FUNCTION_BLOCK REAL2REAL (* Basic Function Block Type *)
  (* Standard: 61499-2 *)
  (* Version 1.0, 2006-11-14, TS, PROFACTOR GmbH *)
  (* Compiler header: package fb.rt.convert; *)
  (* Compiler Java Sun JDK >1.3 *)
  (* Compiler Cpp GNU GCC >3.0 *)
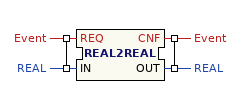
  EVENT_INPUT
    REQ WITH IN; (* Normal Execution Request *)
  END_EVENT
  EVENT_OUTPUT
    CNF WITH OUT; (* Execution Confirmation *)
  END_EVENT
  VAR_INPUT
    IN : REAL; (* Input event qualifier *)
  END_VAR
  VAR_OUTPUT
    OUT : REAL; (* Output event qualifier *)
  END_VAR
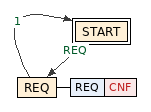
  EC_STATES
    START; (* Initial State *)
    REQ : REQ -> CNF; (* Normal execution *)
  END_STATES
  EC_TRANSITIONS
    START TO REQ := REQ;
    REQ TO START := 1;
  END_TRANSITIONS
  ALGORITHM REQ IN ST: (* Normally executed algorithm *)
OUT:=IN;
  END_ALGORITHM
END_FUNCTION_BLOCK
